{attribute 'qualified_only'}
{attribute 'strict'}
{attribute 'to_string'}
TYPE ERROR_SOURCE_DISPLAY_MODE :
(
	HIDDEN := 0,
	TOP, 
	TOP_AND_ROOT
);
END_TYPE

(* stored: Version 1.1.0.1
   DUT ERROR_SOURCE_DISPLAY_MODE: Id {12200196-fc28-4f0a-bbc7-2eb21d5a35a7} *)
